FUNCTION_BLOCK E_STOP
  (* Version 1.0, 2005-12-19, Goran Cengic, Chalmers *)
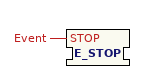
  EVENT_INPUT
    STOP;
  END_EVENT
END_FUNCTION_BLOCK
